// Mitsubishi GX Works2 project: counter3   PLC: Q03UDV

PROGRAM MAIN
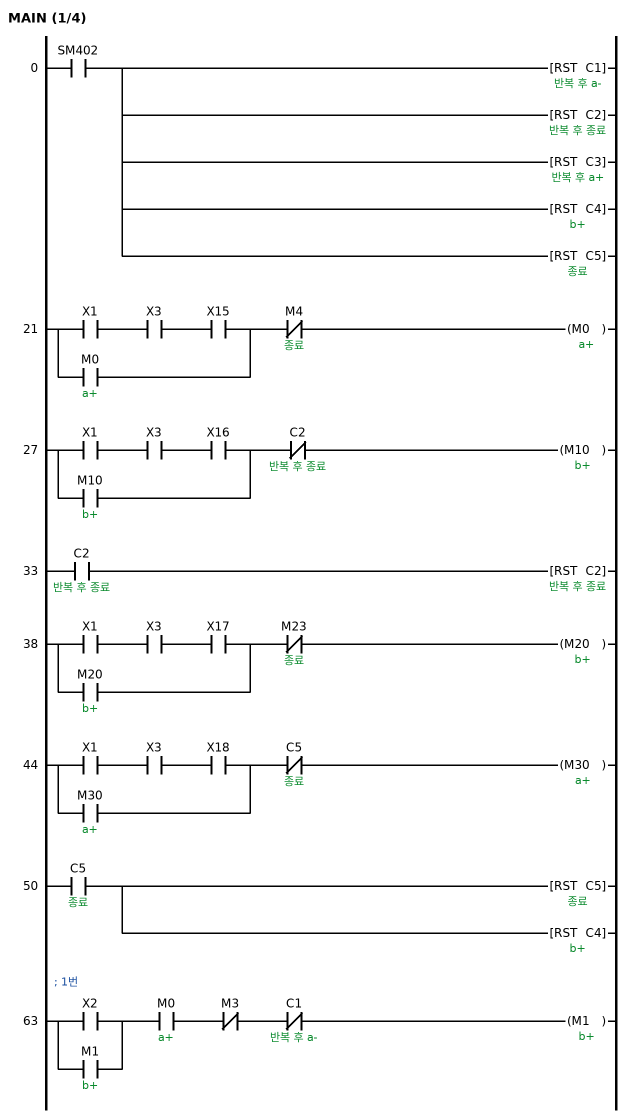
0     LD      SM402
      RST     C1  ; 반복 후 a-
      RST     C2  ; 반복 후 종료
      RST     C3  ; 반복 후 a+
      RST     C4  ; b+
      RST     C5  ; 종료
21    LD      X1
      AND     X3
      AND     X15
      OR      M0  ; a+
      ANI     M4  ; 종료
      OUT     M0  ; a+
27    LD      X1
      AND     X3
      AND     X16
      OR      M10  ; b+
      ANI     C2  ; 반복 후 종료
      OUT     M10  ; b+
33    LD      C2  ; 반복 후 종료
      RST     C2  ; 반복 후 종료
38    LD      X1
      AND     X3
      AND     X17
      OR      M20  ; b+
      ANI     M23  ; 종료
      OUT     M20  ; b+
44    LD      X1
      AND     X3
      AND     X18
      OR      M30  ; a+
      ANI     C5  ; 종료
      OUT     M30  ; a+
50    LD      C5  ; 종료
      RST     C5  ; 종료
      RST     C4  ; b+
; 1번
63    LD      X2
      OR      M1  ; b+
      AND     M0  ; a+
      ANI     M3
      ANI     C1  ; 반복 후 a-
      OUT     M1  ; b+
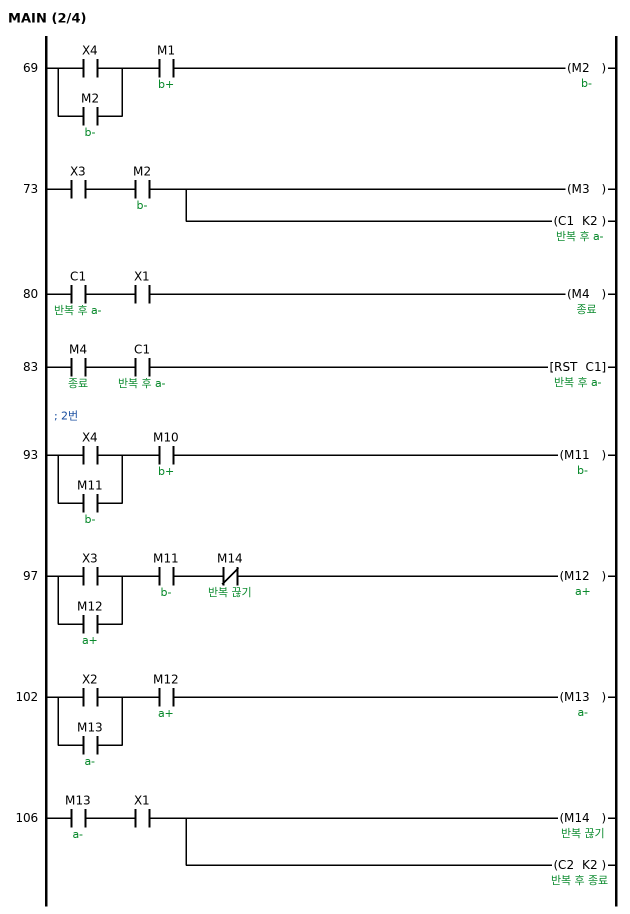
69    LD      X4
      OR      M2  ; b-
      AND     M1  ; b+
      OUT     M2  ; b-
73    LD      X3
      AND     M2  ; b-
      OUT     M3
      OUT     C1 K2  ; 반복 후 a-
80    LD      C1  ; 반복 후 a-
      AND     X1
      OUT     M4  ; 종료
83    LD      M4  ; 종료
      AND     C1  ; 반복 후 a-
      RST     C1  ; 반복 후 a-
; 2번
93    LD      X4
      OR      M11  ; b-
      AND     M10  ; b+
      OUT     M11  ; b-
97    LD      X3
      OR      M12  ; a+
      AND     M11  ; b-
      ANI     M14  ; 반복 끊기
      OUT     M12  ; a+
102   LD      X2
      OR      M13  ; a-
      AND     M12  ; a+
      OUT     M13  ; a-
106   LD      M13  ; a-
      AND     X1
      OUT     M14  ; 반복 끊기
      OUT     C2 K2  ; 반복 후 종료
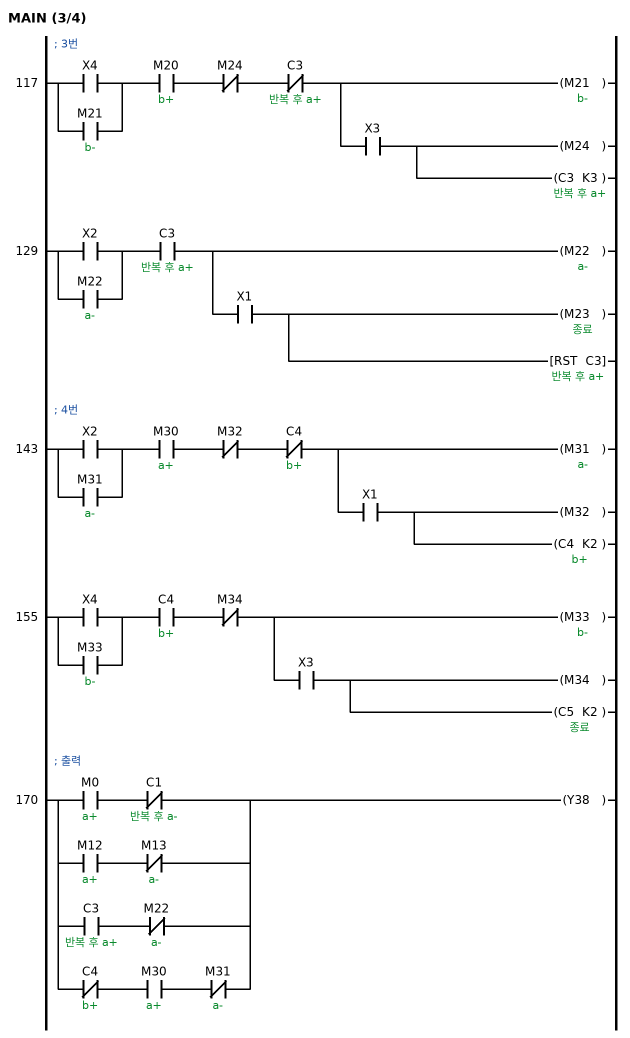
; 3번
117   LD      X4
      OR      M21  ; b-
      AND     M20  ; b+
      ANI     M24
      ANI     C3  ; 반복 후 a+
      OUT     M21  ; b-
      AND     X3
      OUT     M24
      OUT     C3 K3  ; 반복 후 a+
129   LD      X2
      OR      M22  ; a-
      AND     C3  ; 반복 후 a+
      OUT     M22  ; a-
      AND     X1
      OUT     M23  ; 종료
      RST     C3  ; 반복 후 a+
; 4번
143   LD      X2
      OR      M31  ; a-
      AND     M30  ; a+
      ANI     M32
      ANI     C4  ; b+
      OUT     M31  ; a-
      AND     X1
      OUT     M32
      OUT     C4 K2  ; b+
155   LD      X4
      OR      M33  ; b-
      AND     C4  ; b+
      ANI     M34
      OUT     M33  ; b-
      AND     X3
      OUT     M34
      OUT     C5 K2  ; 종료
; 출력
170   LD      M0  ; a+
      ANI     C1  ; 반복 후 a-
      LD      M12  ; a+
      ANI     M13  ; a-
      ORB
      LD      C3  ; 반복 후 a+
      ANI     M22  ; a-
      ORB
      LDI     C4  ; b+
      AND     M30  ; a+
      ANI     M31  ; a-
      ORB
      OUT     Y38
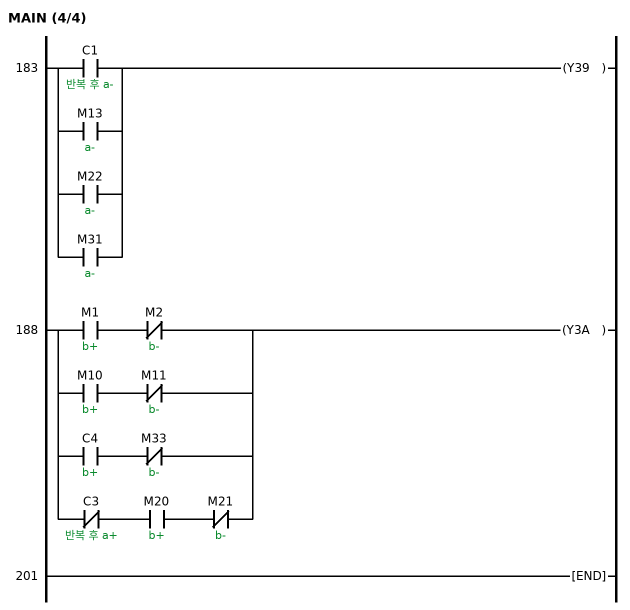
183   LD      C1  ; 반복 후 a-
      OR      M13  ; a-
      OR      M22  ; a-
      OR      M31  ; a-
      OUT     Y39
188   LD      M1  ; b+
      ANI     M2  ; b-
      LD      M10  ; b+
      ANI     M11  ; b-
      ORB
      LD      C4  ; b+
      ANI     M33  ; b-
      ORB
      LDI     C3  ; 반복 후 a+
      AND     M20  ; b+
      ANI     M21  ; b-
      ORB
      OUT     Y3A
201   END
END_PROGRAM
